FUNCTION_BLOCK CAC_Mirror
VAR_INPUT
END_VAR
VAR_OUTPUT
END_VAR
VAR
	Value : REAL;			// from partner's EtherCAT I/O, via WinCC OA
	OutOfRange : BOOL;		// from partner's EtherCAT I/O, via WinCC OA
	Offline: BOOL;			// from partner's EtherCAT I/O, via WinCC OA
	SetInclude : BOOL;		// set on graphics, reset by WinCC OA
	SetExclude : BOOL;		// set on graphics, reset by WinCC OA
	Excluded : BOOL;		// maintained by WinCC OA
	Alarm : BOOL;			// maintained by WinCC OA
	SetIncludeTrig: R_TRIG;	
	SetExcludeTrig: R_TRIG;
END_VAR

VAR_TEMP
	i: INT;	
	modbusReal : ModbusRealWordUnion;
END_VAR


i := GVL.nOutputRegisterIndex;
modbusReal.wordValue[1] := GVL.mb_Output_Registers[i+0];
modbusReal.wordValue[2] := GVL.mb_Output_Registers[i+1];
Value := modbusReal.realValue;
GVL.nOutputRegisterIndex := i+2;


i := GVL.nOutputCoilIndex;
OutOfRange := GVL.mb_Output_Coils[i+0];
Offline := GVL.mb_Output_Coils[i+1];

SetIncludeTrig(CLK:=SetInclude);
IF SetIncludeTrig.Q THEN
	GVL.mb_Output_Coils[i+2] := TRUE;
ELSIF SetInclude AND GVL.mb_Output_Coils[i+2] = 0 THEN
	SetInclude := FALSE;
END_IF

SetExcludeTrig(CLK:=SetExclude);
IF SetExcludeTrig.Q THEN
	GVL.mb_Output_Coils[i+3] := TRUE;
ELSIF SetExclude AND GVL.mb_Output_Coils[i+3] = 0 THEN
	SetExclude := FALSE;
END_IF

Excluded := GVL.mb_Output_Coils[i+4];
Alarm := GVL.mb_Output_Coils[i+5];
GVL.nOutputCoilIndex := i+6;

END_FUNCTION_BLOCK

(* stored: Version 1.1.0.1, ProductVersion 3.1.4024.12
   POU CAC_Mirror: Id {e8b7aef1-2564-48b8-a210-130d2c8d7a76}, SpecialFunc None *)
